FUNCTION_BLOCK FB_VeryBasicMotor IMPLEMENTS I_Axis
VAR_INPUT
	iAnalogInput 	: INT; //Feedback from hardware
	// Scaling of feedback/command values
	fScalingFactor	: LREAL := 1;
END_VAR
VAR_OUTPUT
	iAnalogOutput 	: INT;  //Output to hardware
END_VAR
VAR
	// Disable Analog Output
	bDisableOutput	: BOOL; //Output is disabled
	bJoggingFwd		: BOOL; //Jogging Fwd
	bJoggingBwd		: BOOL; //Jogging bwd
	bMoveAtVelocity	: BOOL;  //moving at velocity
	fCurrentPosition: LREAL;
END_VAR

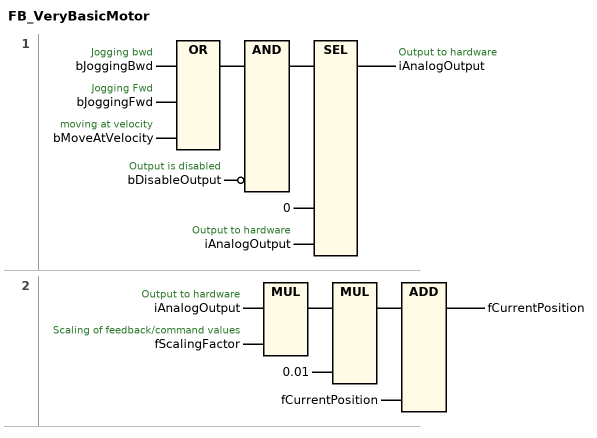
// NETWORK 1
//   bJoggingBwd: Jogging bwd
//   bJoggingFwd: Jogging Fwd
//   bMoveAtVelocity: moving at velocity
//   bDisableOutput: Output is disabled
//   iAnalogOutput: Output to hardware
iAnalogOutput := SEL((bJoggingBwd OR bJoggingFwd OR bMoveAtVelocity) AND NOT bDisableOutput, 0, iAnalogOutput);

// NETWORK 2
//   iAnalogOutput: Output to hardware
//   fScalingFactor: Scaling of feedback/command values
fCurrentPosition := (iAnalogOutput * fScalingFactor) * 0.01 + fCurrentPosition;

METHOD M_Disable : UDINT  //Result of Method
VAR_INPUT
	bDisable	: BOOL; //Input to Method
END_VAR
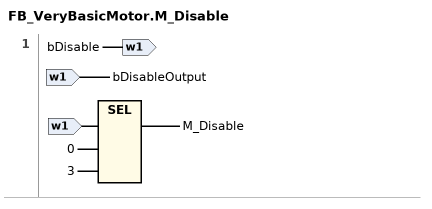
// NETWORK 1
bDisableOutput := bDisable;
M_Disable := SEL(bDisable, 0, 3);
END_METHOD

METHOD M_Enable : UDINT //Method Result
VAR_INPUT
	bEnable	: BOOL;  //Enable Output
END_VAR

VAR
	b1: BOOL;
	b2: BOOL;
END_VAR
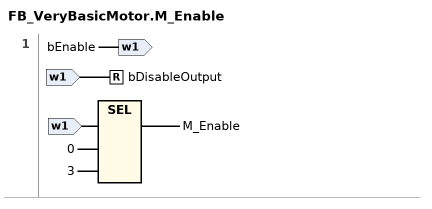
// NETWORK 1
bDisableOutput R= bEnable;
M_Enable := SEL(bEnable, 0, 3);
END_METHOD

METHOD M_HardwareReset : UDINT  //Result of Method Call
VAR_INPUT
	bReset	: BOOL;  //Bit to request hardware reset
END_VAR
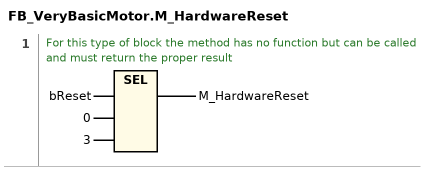
// NETWORK 1
// For this type of block the method has no function but can be called
// and must return the proper result
M_HardwareReset := SEL(bReset, 0, 3);
END_METHOD

METHOD M_Jog : UDINT //Output of block 0 idle 1 busy 3 complete
VAR_INPUT
	bJogFwd	: BOOL;  //Jog fwd command
	bJogBwd	: BOOL; // Jog bwd command
	fJogSpeed	: LREAL;  //speed to jog at
END_VAR

VAR
	
	v1 : LREAL; 
END_VAR
VAR_INST // added by the converter: edge detectors and wires of the graphical bodies
    _w1, _w2 : BOOL;
END_VAR
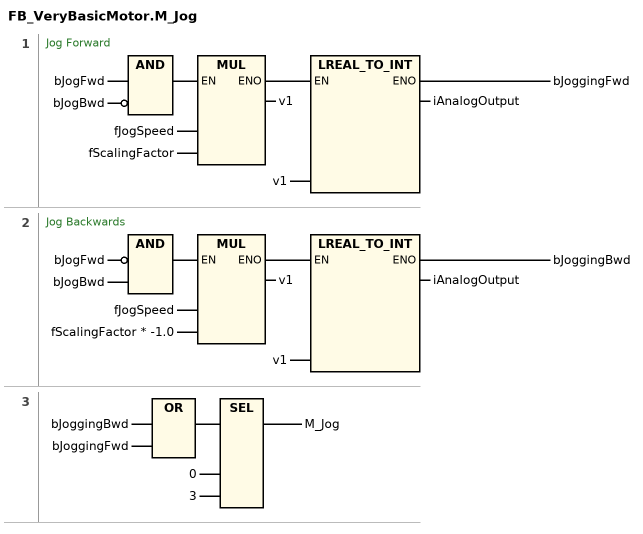
// NETWORK 1
// Jog Forward
_w1 := bJogFwd AND NOT bJogBwd;
IF _w1 THEN v1 := fJogSpeed * fScalingFactor; END_IF
IF _w1 THEN iAnalogOutput := LREAL_TO_INT(v1); END_IF
bJoggingFwd := _w1;

// NETWORK 2
// Jog Backwards
_w2 := NOT bJogFwd AND bJogBwd;
IF _w2 THEN v1 := fJogSpeed * (fScalingFactor * -1.0); END_IF
IF _w2 THEN iAnalogOutput := LREAL_TO_INT(v1); END_IF
bJoggingBwd := _w2;

// NETWORK 3
M_Jog := SEL(bJoggingBwd OR bJoggingFwd, 0, 3);
END_METHOD

METHOD M_Reset : UDINT
VAR_INPUT
	bReset	: BOOL;
END_VAR
END_METHOD

METHOD M_Speed : UDINT
VAR_INPUT
	bMoveVelocity	: BOOL;
	fSpeed	: LREAL;
END_VAR
VAR
	v1:LREAL;
END_VAR
VAR_INST // added by the converter: edge detectors and wires of the graphical bodies
    _w1 : BOOL;
END_VAR
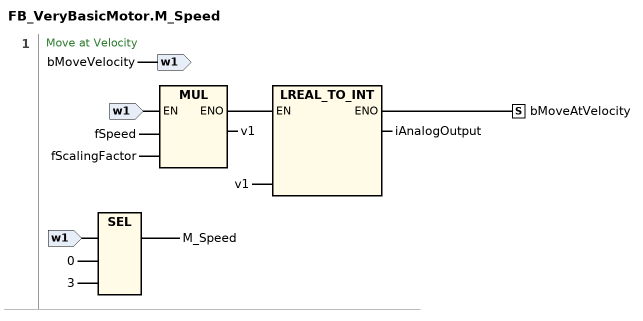
// NETWORK 1
// Move at Velocity
_w1 := bMoveVelocity;
IF _w1 THEN v1 := fSpeed * fScalingFactor; END_IF
IF _w1 THEN iAnalogOutput := LREAL_TO_INT(v1); END_IF
bMoveAtVelocity S= _w1;
M_Speed := SEL(bMoveVelocity, 0, 3);
END_METHOD

METHOD M_Stop : UDINT
VAR_INPUT
	bStop	: BOOL;
END_VAR

VAR

END_VAR
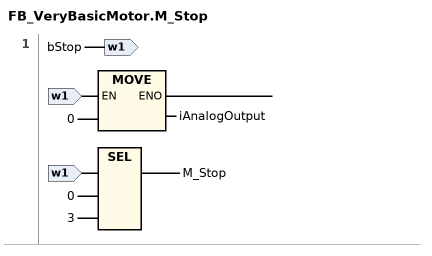
// NETWORK 1
IF bStop THEN iAnalogOutput := 0; END_IF
M_Stop := SEL(bStop, 0, 3);
END_METHOD

PROPERTY P_CurrentPosition : LREAL
GET
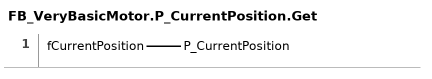
// NETWORK 1
P_CurrentPosition := fCurrentPosition;
END_GET
SET
END_SET
END_PROPERTY

PROPERTY P_CurrentSpeed : LREAL
GET
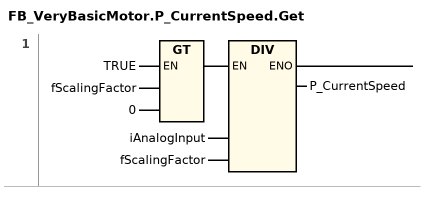
// NETWORK 1
IF fScalingFactor > 0 THEN P_CurrentSpeed := iAnalogInput / fScalingFactor; END_IF
END_GET
SET
END_SET
END_PROPERTY

PROPERTY P_Error : BOOL
GET
END_GET
SET
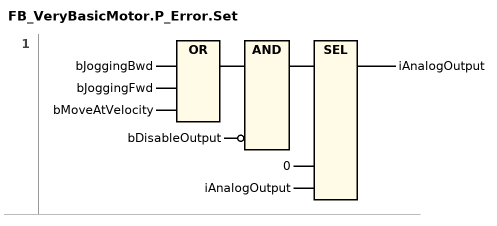
// NETWORK 1
iAnalogOutput := SEL((bJoggingBwd OR bJoggingFwd OR bMoveAtVelocity) AND NOT bDisableOutput, 0, iAnalogOutput);
END_SET
END_PROPERTY

PROPERTY P_ErrorID : UDINT
GET
END_GET
SET
END_SET
END_PROPERTY

PROPERTY P_Ready : BOOL
GET
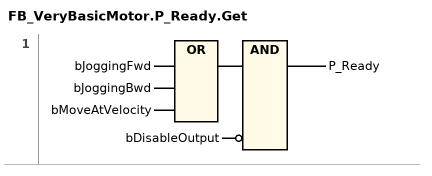
// NETWORK 1
P_Ready := (bJoggingFwd OR bJoggingBwd OR bMoveAtVelocity) AND NOT bDisableOutput;
END_GET
SET
END_SET
END_PROPERTY

END_FUNCTION_BLOCK

(* stored: Version 1.1.0.1, ProductVersion 3.1.4024.11
   POU FB_VeryBasicMotor: Id {6f12638c-2f47-4357-a63b-8be7c08a83d5}, SpecialFunc None
   Method M_Disable: Id {b643319d-248b-44c8-a8f9-af7033ff4419}
   Method M_Enable: Id {a4976f4e-69fa-4142-900f-002fafb6d145}
   Method M_HardwareReset: Id {73cd28bd-514d-4603-bac2-c0d7fe294be1}
   Method M_Jog: Id {b8d91de5-16aa-40e3-bc31-0116ed3cbe19}
   Method M_Reset: Id {272ecb77-e58d-472f-98bd-898020f6258c}
   Method M_Speed: Id {bbf77f1e-a451-4e56-bdd1-db8afd666506}
   Method M_Stop: Id {0a586cb6-49e2-4b8a-a830-bb2d791b9dcf}
   Property P_CurrentPosition: Id {a190ff10-012d-4476-a772-a575bbb37f45}
   Get Get: Id {c8932591-11a1-4c0b-a820-6241c0d6afcb}
   Set Set: Id {87ae23e9-6611-43a3-96b2-90374b55a477}
   Property P_CurrentSpeed: Id {097a0a5c-382f-4bce-905e-01e34343e5b5}
   Get Get: Id {630bc832-89da-4f8d-a89f-8cf95fcb9f98}
   Set Set: Id {ebc5e758-5a2d-499b-9027-4220a4104d0c}
   Property P_Error: Id {6666ecd1-8764-4193-9d33-01b534c0c11b}
   Get Get: Id {b5fc7e2b-a6d8-49fb-b283-41c64c84b5ad}
   Set Set: Id {5aadfaab-eb11-4851-a39d-b4344e969b4b}
   Property P_ErrorID: Id {f6dd5482-01bf-4fbe-a922-3a0519390687}
   Get Get: Id {c10218dd-3bb7-4847-95f8-8a2c6cc9e429}
   Set Set: Id {2b8cf744-0ad9-4055-9977-bfb28ce21745}
   Property P_Ready: Id {1a476de9-9087-422f-ad80-f38999e9f53d}
   Get Get: Id {f51e3981-8e4a-4a94-a18c-7895e3d13aea}
   Set Set: Id {c4cec7dd-40c3-46da-a43f-346e493415e7} *)
